{attribute 'no_explicit_call' := 'Do not call the body - Stick to OOP'}
FUNCTION_BLOCK FB_XTS_Environment EXTENDS FB_CH_Object IMPLEMENTS I_XTS_Environment
VAR
	{attribute 'hide'}
	bInitDone : BOOL ;
	{attribute 'hide'}
	ipXtsSystem : I_XTS_System_Registration;

	fbUtilityEnvironment : Tc3_XTS_Utility.FB_TcIoXtsEnvironment;
	
	//Ethercat Diagnostic of all XTS Motors
	fbXtsEtherCatDiag		: FB_XtsEtherCatDiag(	ipUtilityEnvironmentv 				:=  fbUtilityEnvironment,
													bCheckIfTc3EventloggerIsSelected 	:= XtsParameterlist.B_MSG_IF_TC3EVENTLOGGER_IS_NOT_DEFAULT);
	
	{attribute 'hide'}
	fbXtsEnvironmentVisu : Tc3_XTS_Utility.FB_XtsEnvironmentVisu;
		
END_VAR

METHOD FB_init : BOOL
VAR_INPUT
	bInitRetains : BOOL; // if TRUE, the retain variables are initialized (warm start / cold start)
	bInCopyCode : BOOL;  // if TRUE, the instance afterwards gets moved into the copy code (online change)

	ipXtsSystem : I_XTS_System_Registration; //Interface to XTS system object	
END_VAR
VAR_INST
	{attribute 'hide'}
	bFBInitCalledOnce : BOOL; //Do the following code once during start up and not during onlinechange
END_VAR
//Do the following code once during start up and not during onlinechange
IF NOT bFBInitCalledOnce THEN 
	
	//Regristrate object in System
	IF ipXtsSystem <> 0 THEN
		ipXtsSystem.LinkEnvironment(THIS^);
		THIS^.ipXtsSystem := ipXtsSystem;
	END_IF



END_IF

bFBInitCalledOnce := TRUE;
END_METHOD

{warning 'add property implementation'}
{attribute 'monitoring':='call'}
PROPERTY HR : HRESULT
GET
HR := S_OK;
END_GET
END_PROPERTY

METHOD Initialize : HRESULT
VAR 
	hr : HRESULT;
END_VAR
IF NOT THIS^.bInitDone THEN
	Initialize := S_PENDING;	

	//Enable init Info Server if needed
	fbUtilityEnvironment.P_XtsEnvironmentConfiguration.bEnableInitInfoServer := TRUE;

	//Enable init CA Group if needed
	fbUtilityEnvironment.P_XtsEnvironmentConfiguration.bEnableInitCaGroup := TRUE;

	IF NOT fbUtilityEnvironment.P_IsInitialized THEN	
		//Start init
		fbUtilityEnvironment.Init(bExecute := TRUE); 
		hr := GetMostSignificant(hr, S_PENDING);	
 	ELSE
		//Stop init
		fbUtilityEnvironment.Init(bExecute := FALSE);
	END_IF
	
	// Link data Pointer 
	fbXtsEnvironmentVisu(ipTcIoXtsEnvironment:=UtilityEnvirement);

	// Ethercat Diagnostic of all XTS Motors
	hr := GetMostSignificant(hr, fbXtsEtherCatDiag.Initialize());
	

	THIS^.bInitDone  :=  hr = S_OK;
END_IF

Initialize := hr;
END_METHOD

{attribute 'monitoring':='call'}
PROPERTY TrackIsRing : BOOL
GET
IF fbUtilityEnvironment.P_IsInitialized THEN
	TrackIsRing := fbUtilityEnvironment.Mc2CaGroup(1).GetRailIsRing();
END_IF
END_GET
END_PROPERTY

{attribute 'monitoring':='call'}
PROPERTY TrackLength : LREAL
GET
IF fbUtilityEnvironment.P_IsInitialized THEN
	TrackLength := fbUtilityEnvironment.Mc2CaGroup(1).GetRailLength();
END_IF
END_GET
END_PROPERTY

METHOD Update : HRESULT
VAR
	hr : HRESULT;
END_VAR

fbXtsEtherCatDiag.Update();

fbXtsEnvironmentVisu.Cycle();

Update:= hr;
END_METHOD

PROPERTY UtilityEnvirement : Tc3_XTS_Utility.I_TcIoXtsEnvironment
GET
//Interface to envirement
UtilityEnvirement := fbUtilityEnvironment;
END_GET
END_PROPERTY

END_FUNCTION_BLOCK

(* stored: Version 1.1.0.1, ProductVersion 3.1.4024.12
   POU FB_XTS_Environment: Id {a8afa6a2-387c-4b6e-9be2-2721f7668e6b}, SpecialFunc None
   Method FB_init: Id {93d2d8fa-7888-47d9-ae7c-4547c74b0ffa}
   Property HR: Id {1aeed165-c0b0-44f5-ad1d-c9c5538bc734}
   Get Get: Id {5822a1eb-9a43-4828-929e-0f8351589bc4}
   Method Initialize: Id {7cd9bb8a-718f-430d-9839-512439f8bc63}
   Property TrackIsRing: Id {24b8be3c-88b3-4d84-8780-5184e661106f}
   Get Get: Id {2537b9e8-b626-449a-ba90-9f59377c75f6}
   Property TrackLength: Id {7be4b154-e932-4cd8-beb2-5b72757cfd1e}
   Get Get: Id {0b5e46ca-1791-4ddd-87d2-a3225362ce10}
   Method Update: Id {84f7e194-e354-4685-a40e-bbd23c57553a}
   Property UtilityEnvirement: Id {cfb048a9-88dd-4d21-8adb-997f876cb0e4}
   Get Get: Id {4e7a3925-6766-42f7-b653-fba6145e43da} *)
